Universal Robots URScript: admittance.script

def song():
  global _hidden_verificationVariable=0
  set_tcp(p[0.028210348281514253, -0.09610723587300697, -0.09969041498611403, 0.0, 0.0, 0.0])
  set_standard_analog_input_domain(0, 1)
  set_standard_analog_input_domain(1, 1)
  set_tool_analog_input_domain(0, 1)
  set_tool_analog_input_domain(1, 1)
  set_analog_outputdomain(0, 0)
  set_analog_outputdomain(1, 0)
  set_input_actions_to_default()
  set_tool_communication(False, 115200, 0, 1, 1.5, 3.5)
  set_tool_output_mode(0)
  set_tool_digital_output_mode(0, 1)
  set_tool_digital_output_mode(1, 1)
  set_tool_voltage(0)
  set_target_payload(0.260000, [0.050000, -0.008000, 0.024000], [0.000163, 0.000163, 0.000163, 0.000000, 0.000000, 0.000000])
  set_safety_mode_transition_hardness(1)
  set_gravity([0.0, 0.0, 9.82])
  global Plane_1=p[0.32571614183608727, 0.7933870146316717, 0.11820742021636722, -2.208244884171713, -0.24738609815952348, -1.9195085473101943]
  global Plane_2=p[0.3436052139151623, 0.7478032414335104, 0.10077839665899768, 2.768545736097797, 0.1284831553507919, 1.3672805628273381]
  global Plane_3=p[0.31945151854627996, 0.6757990361168175, 0.09459088830114093, 2.7301760593116526, -0.049483824131046385, 1.4252239353300047]
  global Plane_4=p[0.3372257363094211, 0.6222230974198586, 0.07001667903587716, 2.621672423508307, -0.12240385890263918, 1.4373011913128484]
  # begin: URCap Installation Node
  #   Source: External Control, 1.0.5, FZI Research Center for Information Technology
  #   Type: External Control
  # end: URCap Installation Node
  # begin: URCap Installation Node
  #   Source: External Control, 1.0.5, FZI Research Center for Information Technology
  #   Type: External Control
  # end: URCap Installation Node
  popup("Started song()")
  textmsg("RUN")
  global _event_flag = 0

  global a_bow_poses = struct(
    tip_p=[.473129539189, .413197423330, .256308427905, -1.460522581833, -2.310115543652, 1.445803824327],
    frog_p=[.300717266074, .793568239540, .099710283103, -1.543522183454, -2.354885618328, 1.346770272474]
  )

  global d_bow_poses = struct(
    tip_p=[.340413993945, .280157415162, .176342071758, -1.614553612482, -2.044810993523, 1.042279199535],
    frog_p=[.302785064368, .749849181019, .117254426008, -1.664082298752, -2.084265434693, 1.037965163360]
  )

  global g_bow_poses = struct(
    tip_p=[.162016291992, .201320984957, .059414774157, -1.929772636560, -1.931323067217, .555055912517],
    frog_p=[.281203376642, .681662588607, .104672526365, -1.812194031755, -1.940153681829, .493747597283]
  )

  global c_bow_poses = struct(
    tip_p=[.079815569355, .285182178102, -.086654726588, -1.819646014269, -1.658258006768, .180930717120],
    frog_p=[.256662516098, .610082591416, .062624387196, -1.743236422252, -1.524514092756, .163823228357]
  )

  # ---- Force-control & lever-arm parameters (tune these) ----
  global r_tool = [0.0, 0.6096, 0.0]    # [x,y,z] in meters (tool frame). Set this from frog TCP -> contact point measurement.
  global target_force = 0.5           # desired normal force at contact (N) — tune
  global admittance_gain = 0.002      # dz = gain * (target - measured); start small
  global max_offset = 0.01            # max Z correction per step (m)
  global control_period = 0.02        # seconds per control step
  global servoj_acc = 0.1
  global servoj_vel = 0.2
  global fuse_alpha = 0.8             # weight for linear Fz projection vs torque-derived estimate
  global orient_comp_gain = 0.0008    # small orientation correction gain (rad per Nm)
  # ----------------------------------------------------------

  def ease_scale(note_dur):
    if note_dur > 3:
      note_dur = 3
    end
    return (1.0 - cos(3.14159265359 * note_dur / 3.0)) / 2.0
  end

  # ------------------ Vector utilities ------------------
  def dot(a, b):
    return a[0]*b[0] + a[1]*b[1] + a[2]*b[2]
  end

  def cross(a, b):
    return [ a[1]*b[2] - a[2]*b[1],
             a[2]*b[0] - a[0]*b[2],
             a[0]*b[1] - a[1]*b[0] ]
  end
  # ------------------------------------------------------

  # ---------- compute unit tool-Z in base frame ----------
  def get_tool_z_hat():
    local tcp = get_actual_tcp_pose()   # base-frame pose
    local zpt = pose_trans(tcp, p[0,0,0.01,0,0,0])  # 1cm along tool Z in base frame
    local zd = [zpt[0]-tcp[0], zpt[1]-tcp[1], zpt[2]-tcp[2]]
    local n = norm(zd)
    if n == 0:
      return [0,0,1]
    end
    return [zd[0]/n, zd[1]/n, zd[2]/n]
  end
  # -------------------------------------------------------

  # ---------- transform r_tool (tool frame) to base frame -------
  def r_tool_to_base(r_tool_param):
    local tcp = get_actual_tcp_pose()
    local contact_pose = pose_trans(tcp, p[r_tool_param[0], r_tool_param[1], r_tool_param[2], 0,0,0])
    return [contact_pose[0]-tcp[0], contact_pose[1]-tcp[1], contact_pose[2]-tcp[2]]
  end
  # ---------------------------------------------------------------

  # ---------- measure & fuse Fz estimate ----------
  def measure_fused_Fz_and_torque():
    # returns a list: [Fz_fused (N), [Tx, Ty, Tz] (Nm)]
    local wrench = get_tcp_force()   # [Fx,Fy,Fz, Tx,Ty,Tz] in base frame
    local F_tcp = [wrench[0], wrench[1], wrench[2]]
    local T_tcp = [wrench[3], wrench[4], wrench[5]]

    # compute tool z_hat and project linear force onto it
    local z_hat = get_tool_z_hat()
    local Fz_proj = dot(F_tcp, z_hat)

    # torque-derived estimate: assume F ≈ Fz * z_hat and tau ≈ r_base x (Fz * z_hat)
    local r_base = r_tool_to_base(r_tool)
    local r_cross_z = cross(r_base, z_hat)
    local denom = dot(r_cross_z, r_cross_z)
    local Fz_from_tau = 0.0
    if denom > 1e-8:
      Fz_from_tau = dot(T_tcp, r_cross_z) / denom
    else:
      Fz_from_tau = Fz_proj   # fallback when lever arm geometry is degenerate
    end

    # fuse (weighted)
    local Fz_fused = fuse_alpha * Fz_proj + (1.0 - fuse_alpha) * Fz_from_tau

    return [Fz_fused, T_tcp[0], T_tcp[1], T_tcp[2]]
  end
  # ----------------------------------------------------

    # ---------- orientation correction (small) ----------
    def orientation_correction(T_tcp_param, Fz_fused_param):
    # return small rotation [rx, ry, 0] in radians to reduce Tx, Ty
      local rx = 0.0
      local ry = 0.0

      # define abs manually
      if Fz_fused_param >= 0.0:
          local absFz = Fz_fused_param
      else:
          local absFz = -Fz_fused_param
      end

      if absFz > 0.2:
          # simple proportional: torque about X -> rotate around Y, torque about Y -> rotate around X
          rx = -orient_comp_gain * T_tcp_param[1] / (absFz + 1e-6)
          ry = orient_comp_gain * T_tcp_param[0] / (absFz + 1e-6)

          # clamp small rotation magnitudes to safe range
          if rx > 0.05:
          rx = 0.05
          elif rx < -0.05:
          rx = -0.05
          end

          if ry > 0.05:
          ry = 0.05
          elif ry < -0.05:
          ry = -0.05
          end
      end

      local rot_vec = [rx, ry, 0.0]
      return rot_vec
    end
    # ----------------------------------------------------


  # ---------- measure force along tool Z (public helper) ----------
  def measure_force_along_tool_z():
    local res = measure_fused_Fz_and_torque()
    local Fz = res[0]
    return Fz
  end
  # ----------------------------------------------------

  # ---------- New bow implementation with admittance-style Z correction ----------
  def bow(bow_dir, note_dur, bow_poses):
    if note_dur > 3:
      note_dur = 3
    end

    local dist_scale = ease_scale(note_dur)

    local tip_p = bow_poses.tip_p
    local frog_p = bow_poses.frog_p

    local tcp_pose = get_actual_tcp_pose()
    local start_p = [tcp_pose[0], tcp_pose[1], tcp_pose[2], tcp_pose[3], tcp_pose[4], tcp_pose[5]]
    local end_p = frog_p

    local direction_vector = (tip_p - frog_p) / norm(tip_p - frog_p)
    local t_dir = -1
    local target_dist = dist_scale * norm(tip_p - frog_p)

    if bow_dir:
      end_p = tip_p
      t_dir = 1
    end

    global ending_spot = end_p

    if (norm(end_p - start_p) >= target_dist):
      end_p = start_p + t_dir * direction_vector * target_dist
    end

    # compute time/steps
    local total_time = note_dur
    if total_time <= 0.0:
      total_time = control_period
    end
    local steps = round(total_time / control_period)
    if steps < 1:
      steps = 1
    end

    local step_vec = (end_p - start_p) / steps

    local i = 1
    while i <= steps:
      # desired interpolated pose in base frame
      local interp = start_p + step_vec * i

      textmsg("Run")

      # measure fused Fz and torque
      local res2 = measure_fused_Fz_and_torque()
      textmsg("Oranges")
      local Fz = res2[0]
      local T_tcp = [res2[1], res2[2], res2[3]]

      # compute dz correction (admittance)
      local error = target_force - Fz
      local dz = admittance_gain * error

      # clamp dz
      if dz > max_offset:
        dz = max_offset
      elif dz < -max_offset:
        dz = -max_offset
      end

      # optionally scale dz by lever-position along bow: compute fraction along bow axis (0..1)
      local A = frog_p
      local bow_vec = tip_p - frog_p
      local frac = 0.0
      local denom = dot(bow_vec, bow_vec)
      if denom > 1e-8:
        frac = dot(interp - A, bow_vec) / denom
      end
      # clamp frac 0..1
      if frac < 0.0:
        frac = 0.0
      elif frac > 1.0:
        frac = 1.0
      end

      textmsg("yellow")

      # lever scaling: when closer to tip (frac near 1), larger lever -> scale correction down
      local lever_scale = 1.0 - 0.5 * frac   # tune this mapping if desired

      local dz_scaled = dz * lever_scale

      textmsg("purple")

      # apply dz relative to TCP
      local base_pose_for_target = p[interp[0], interp[1], interp[2], interp[3], interp[4], interp[5]]
      local target_pose = pose_trans(base_pose_for_target, p[0,0,dz_scaled,0,0,0])

      # small orientation correction from torque
      local rot = orientation_correction(T_tcp, Fz)
      if (rot[0] != 0.0) or (rot[1] != 0.0):
        target_pose = pose_trans(target_pose, p[0,0,0, rot[0], rot[1], rot[2]])
      end


      # command the small step using servoj for smoothness
      local target_q = get_inverse_kin(target_pose)
      servoj(target_q, servoj_acc, servoj_vel, control_period, 0.05, 300)
      textmsg("rum")
      sync()
      i = i + 1
    end
  end
  # ----------------------------------------------------

  def stay():
    stopj(2.5)
    sleep(0.025)
  end

  def a_bow(bow_dir, note_dur):
    _event_flag = 1  # START a_bow
    write_output_integer_register(0, _event_flag)
    write_output_integer_register(1, bow_dir)
    bow(bow_dir, note_dur, a_bow_poses)
    _event_flag = 2  # END a_bow
    write_output_integer_register(0, _event_flag)
  end

  def d_bow(bow_dir, note_dur):
    _event_flag = 3  # START d_bow
    write_output_integer_register(1, bow_dir)
    write_output_integer_register(0, _event_flag)
    bow(bow_dir, note_dur, d_bow_poses)
    _event_flag = 4  # END d_bow
    write_output_integer_register(0, _event_flag)
  end

  def g_bow(bow_dir, note_dur):
    _event_flag = 5  # START g_bow
    write_output_integer_register(1, bow_dir)
    write_output_integer_register(0, _event_flag)
    bow(bow_dir, note_dur, g_bow_poses)
    _event_flag = 6  # END g_bow
    write_output_integer_register(0, _event_flag)
  end

  def c_bow(bow_dir, note_dur):
    _event_flag = 7  # START c_bow
    write_output_integer_register(1, bow_dir)
    write_output_integer_register(0, _event_flag)
    bow(bow_dir, note_dur, c_bow_poses)
    _event_flag = 8  # END c_bow
    write_output_integer_register(0, _event_flag)
  end

  def round(n):
    local int_part = floor(n)
    if (n - int_part) >= 0.5:
      return int_part + 1
    else:
      return int_part
    end
  end

  def min(a, b):
    if a < b:
      return a
    else:
      return b
    end
  end

  def max(a, b):
    if a > b:
      return a
    else:
      return b
    end
  end

  # NOTE: dot already defined above; preserved.

  def string_crossing(start_bow_poses, end_bow_poses, next_dir):
    # we first find the curr position
    local tcp_pose = get_actual_tcp_pose()
    local start_p = [tcp_pose[0], tcp_pose[1], tcp_pose[2], tcp_pose[3], tcp_pose[4], tcp_pose[5]]

    local out = [0.89583677, 0.04158029, 0.44243367, 0, 0, 0]
    local step1 = start_p + out * 0.03

    movep(p[step1[0], step1[1], step1[2], start_p[3], start_p[4], start_p[5]])
    movep(p[step1[0], step1[1], step1[2], d_bow_poses.frog_p[3], d_bow_poses.frog_p[4], d_bow_poses.frog_p[5]])
    sync()

    tcp_pose = get_actual_tcp_pose()
    start_p = [tcp_pose[0], tcp_pose[1], tcp_pose[2], tcp_pose[3], tcp_pose[4], tcp_pose[5]]
    local bow_vec = end_bow_poses.tip_p - end_bow_poses.frog_p
    local direction_vector = bow_vec / norm(bow_vec)
    local A = end_bow_poses.tip_p
    local target_pose = dot(start_p - A, direction_vector) / dot(direction_vector, direction_vector) * direction_vector + A

    movep(p[target_pose[0], target_pose[1], target_pose[2], target_pose[3], target_pose[4], target_pose[5]], v=3.67)
    # sync()

  end

  def a_to_d(next_dir=0):
    _event_flag = 101
    write_output_integer_register(0, _event_flag)
    string_crossing(a_bow_poses, d_bow_poses, next_dir)
    _event_flag = 102
    write_output_integer_register(0, _event_flag)
  end

  def a_to_g(next_dir=0):
    _event_flag = 109
    write_output_integer_register(0, _event_flag)
    string_crossing(a_bow_poses, g_bow_poses, next_dir)
    _event_flag = 110
    write_output_integer_register(0, _event_flag)
  end

  def d_to_a(next_dir=0):
    _event_flag = 103
    write_output_integer_register(0, _event_flag)
    string_crossing(d_bow_poses, a_bow_poses, next_dir)
    _event_flag = 104
    write_output_integer_register(0, _event_flag)
  end

  def d_to_g(next_dir=0):
    _event_flag = 105
    write_output_integer_register(0, _event_flag)
    string_crossing(d_bow_poses, g_bow_poses, next_dir)
    _event_flag = 106
    write_output_integer_register(0, _event_flag)
  end

  def d_to_c(next_dir=0):
    _event_flag = 113
    write_output_integer_register(0, _event_flag)
    string_crossing(d_bow_poses, c_bow_poses, next_dir)
    _event_flag = 114
    write_output_integer_register(0, _event_flag)
  end

  def g_to_a(next_dir=0):
    _event_flag = 111
    write_output_integer_register(0, _event_flag)
    string_crossing(g_bow_poses, a_bow_poses, next_dir)
    _event_flag = 112
    write_output_integer_register(0, _event_flag)
  end

  def g_to_d(next_dir=0):
    _event_flag = 107
    write_output_integer_register(0, _event_flag)
    string_crossing(g_bow_poses, d_bow_poses, next_dir)
    _event_flag = 108
    write_output_integer_register(0, _event_flag)
  end

  def g_to_c(next_dir=0):
    _event_flag = 117
    write_output_integer_register(0, _event_flag)
    string_crossing(g_bow_poses, c_bow_poses, next_dir)
    _event_flag = 118
    write_output_integer_register(0, _event_flag)
  end

  def c_to_d(next_dir=0):
    _event_flag = 115
    write_output_integer_register(0, _event_flag)
    string_crossing(c_bow_poses, d_bow_poses, next_dir)
    _event_flag = 116
    write_output_integer_register(0, _event_flag)
  end

  def c_to_g(next_dir=0):
    _event_flag = 119
    write_output_integer_register(0, _event_flag)
    string_crossing(c_bow_poses, g_bow_poses, next_dir)
    _event_flag = 120
    write_output_integer_register(0, _event_flag)
  end

  stay()
  stay()
  # $$$ CODE HERE $$$  # (you can call a_bow/d_bow/g_bow/c_bow or the crossing functions here)
  d_bow(1, 1.9979166666666666)
  stay()
  d_bow(1, 1.9979166666666666)
  stay()

end

song()
